(* IEC 61131-3 sources: programs/VI-54/VI-54_20171205/VI-54_20171205/Stations/PLC_VI54/VI-54_171014/Class/Camera_Master, 1 file *)

(* ---- Camera_Master.st ---- *)
(*!
<Class
	Name               = "Camera_Master"
	Revision           = "2.0"
	RealtimeTask       = "false"
	CyclicTask         = "false"
	BackgroundTask     = "false"
	Sigmatek           = "false"
	OSInterface        = "false"
	HighPriority       = "false"
	Automatic          = "false"
	UpdateMode         = "Prescan"
	SharedCommandTable = "true"
	Objectsize         = "(630,120)">
	<Channels>
		<Server Name="DataCompleted" Visualized="true" Initialize="false" WriteProtected="false" Retentive="false"/>
		<Server Name="IsOnline" Visualized="true" Initialize="false" WriteProtected="true" Retentive="false"/>
		<Server Name="NbrOfTriggers" Visualized="true" Initialize="false" WriteProtected="true" Retentive="false"/>
		<Server Name="SendCommand" Visualized="true" Initialize="false" WriteProtected="false" Retentive="false"/>
		<Server Name="TmrNewConnection" Visualized="true" Initialize="true" WriteProtected="false" Retentive="File"/>
		<Client Name="_TCPIP_CLIENT2" Required="true" Internal="true"/>
		<Client Name="cPort" Required="true" Internal="false" Comment="port number ... must be connected or initialized"/>
		<Client Name="iFc_Trigger" Required="true" Internal="false"/>
		<Client Name="IpAdres" Required="true" Internal="true"/>
	</Channels>
	<Separators>
		<Servers>
			<SepChn Position="3"/>
			<SepChn Position="5"/>
		</Servers>
	</Separators>
	<Network Name="Camera_Master">
		<!-- List of Components in this network -->
		<Components>
			<Object
				Name       = "_base"
				Class      = "MachineBase"
				Position   = "(218,120)"
				Visualized = "true">
				<Channels>
					<Server Name="ObjectServer"/>
					<Server Name="RunningMode"/>
					<Server Name="Stepper"/>
				</Channels>
			</Object>
			<Object
				Name           = "_TCPIP_CLIENT2"
				Class          = "_TCPIP_CLIENT"
				Position       = "(210,660)"
				Visualized     = "false"
				CyclicTime     = "10 ms"
				BackgroundTime = "always">
				<Channels>
					<Server Name="Control"/>
					<Server Name="SemaName01"/>
					<Server Name="SemaName02"/>
					<Server Name="TaskName"/>
					<Client Name="cConfig"/>
					<Client Name="cMaxConnections" Value="0"/>
					<Client Name="co_MultiTask"/>
					<Client Name="co_SigCLib"/>
					<Client Name="co_StdLib"/>
					<Client Name="co_Task"/>
					<Client Name="cPort" Value="500"/>
					<Client Name="cSizeOfTXBuffer"/>
				</Channels>
			</Object>
			<Object
				Name       = "IpAdres"
				Class      = "StringRAM"
				Position   = "(210,420)"
				Visualized = "true"
				Remotely   = "true">
				<Channels>
					<Server Name="Data" Value="&quot;10.10.150.26&quot;"/>
					<Client Name="SingleRealloc" Value="1"/>
					<Client Name="UseFile"/>
				</Channels>
			</Object>
		</Components>
		<Comments>
		</Comments>
		<!-- List of Connections in this network -->
		<Connections>
			<Connection Source="this.ObjectServer" Destination="_base.ObjectServer" Vertices="(1006,210),(834,210),"/>
			<Connection Source="this.Stepper" Destination="_base.Stepper" Vertices="(1006,270),(834,270),"/>
			<Connection Source="this.RunningMode" Destination="_base.RunningMode" Vertices="(1006,330),(834,330),"/>
			<Connection Source="this.IpAdres" Destination="IpAdres.Data"/>
			<Connection Source="this._TCPIP_CLIENT2" Destination="_TCPIP_CLIENT2.Control"/>
			<Connection Source="_TCPIP_CLIENT2.cPort" Destination="this.cPort" Vertices="(210,750),(38,390),"/>
		</Connections>
		<!-- Headerfiles -->
		<Options>
		</Options>
	</Network>
</Class>
*)
#pragma using MachineBase

Camera_Master : CLASS
: MachineBase
	TYPE
	  IpAdrStr : ARRAY [0..15] OF CHAR;
	  SendCommands :  //! <Type Public="true" Name="SendCommands"/>
	  (
	    eNoCommand,
	    eReboot,
	    eRestart,
	    eTrigger
	  )$UDINT;
#pragma pack(push, 1)
	  SendStr : STRUCT
	    HeartBeat : BOOL;
	    Command : SendCommands;
	  END_STRUCT;
#pragma pack(pop)
	END_TYPE
  //Servers:
	IsOnline 	: SvrCh_DINT;
	NbrOfTriggers 	: SvrCh_DINT;
	TmrNewConnection 	: SvrCh_UDINT;
	DataCompleted 	: SvrCh_DINT;
	SendCommand 	: SvrCh_SendCommands_PTofCls_Camera_Master;
  //Clients:
	IpAdres 	: CltChCmd_StringRAM;
	cPort 	: CltCh_DINT;
	_TCPIP_CLIENT2 	: CltChCmd__TCPIP_CLIENT;
	iFc_Trigger 	: CltChCmd_ProductTrigger;
  //Variables:
		Handle 	: DINT;
		Adress_TCP 	: IpAdrStr;
		CameraDataStr 	: CameraData;
		TmrDelay 	: UDINT;
		TmrHeartBeat 	: UDINT;
		CameraBits : BDINT
		[
		  1 SendStr,
		];

		SendData 	: SendStr;
  //Functions:

	FUNCTION VIRTUAL GLOBAL MyCyTask;

	FUNCTION GLOBAL MyCallBack
		VAR_INPUT
			pData 	: ^void;
			udSize 	: UDINT;
		END_VAR;

	FUNCTION GLOBAL GetData
		VAR_OUTPUT
			Ptr 	: CameraData;
		END_VAR;

	FUNCTION GLOBAL ResetData;

	FUNCTION GLOBAL gmSendData
		VAR_INPUT
			Data 	: ^void;
		END_VAR
		VAR_OUTPUT
			Retcode 	: BOOL;
		END_VAR;

	FUNCTION GLOBAL gmHeartBeat;

	FUNCTION GLOBAL gmTrigger;

	FUNCTION VIRTUAL GLOBAL SendCommand::Write
		VAR_INPUT
			input (EAX) 	: Camera_Master::SendCommands;
		END_VAR
		VAR_OUTPUT
			result (EAX) 	: Camera_Master::SendCommands;
		END_VAR;
  //Tables:
	FUNCTION @STD
		VAR_OUTPUT
			ret_code	: CONFSTATES;
		END_VAR;
	FUNCTION GLOBAL TAB @CT_;
END_CLASS;

#pragma using _TCPIP_CLIENT
#pragma using StringRAM
#pragma usingLtd ProductTrigger

FUNCTION VIRTUAL GLOBAL Camera_Master::MyCyTask

  _TCPIP_CLIENT2.CyWork(EAX:= 0);
  IsOnline := _TCPIP_CLIENT2.IsConnected(dHandle:= Handle);

  // Open methodes
  gmTrigger();
  gmHeartBeat();

  // Check for sending data
  if CameraBits.SendStr = true then
    if gmSendData(Data:= #SendData) = true then
      CameraBits.SendStr := False;
    end_if;
  end_if;

  case Stepper of
  00: // Check communication
    if IsOnline = false then
      Stepper += 1;
    end_if;

  01: // Make connection
    IpAdres.ReadDataOff(udOff:= 0, pData:= #Adress_TCP$Usint, udMax := sizeof(IpAdrStr));
    Adress_TCP[15] := cNul;
    Handle := _TCPIP_CLIENT2.AddConnection( pIPAddress    := "10.10.150.26",
                                            pCallbackThis := this,
                                            pCallbackMeth := #MyCallBack(),
                                            udTimeout     := 0);
    TmrDelay := ops.tAbsolute;
    Stepper += 1;

  02: // Check online state
    if IsOnline > 0 then
      TmrDelay := ops.tAbsolute;
    elsif (ops.tAbsolute - TmrDelay) >= TmrNewConnection then
      Stepper -= 1;
    end_if;
  end_case;

END_FUNCTION

FUNCTION GLOBAL Camera_Master::MyCallBack
	VAR_INPUT
		pData 	: ^void;
		udSize 	: UDINT;
	END_VAR

  // Set data into array
  _memset(dest:= #CameraDataStr, usByte:= 0, cntr:= sizeof(CameraData));
  _memcpy(ptr1:= #CameraDataStr, ptr2:= pData, cntr:= sizeof(CameraData));

  // Set bit that we receive new data
  DataCompleted := 1;

END_FUNCTION

FUNCTION GLOBAL Camera_Master::GetData
	VAR_OUTPUT
		Ptr 	: CameraData;
	END_VAR

  Ptr := CameraDataStr;

  // Reset data after reading
  ResetData();

END_FUNCTION

FUNCTION GLOBAL Camera_Master::ResetData

  // Reset all the data
  DataCompleted     := 0;

  // Reset pointer
  _memset(dest:= #CameraDataStr, usByte:= 0, cntr:= sizeof(CameraData));

END_FUNCTION

FUNCTION GLOBAL Camera_Master::gmHeartBeat

  // Every second a heartbeat
  if (ops.tAbsolute - TmrHeartBeat) >= 1000 then
    SendData.HeartBeat  := (SendData.HeartBeat XOR 1);
    CameraBits.SendStr  := true;
    TmrHeartBeat        := ops.tAbsolute;
  end_if;

END_FUNCTION

FUNCTION GLOBAL Camera_Master::gmTrigger

  // Set trigger offset
  iFc_Trigger.SetTriggerOffset(State:= (RecipePtr^.Camera.TriggerOffset * cIntUnitsTo_mm));

  // Check trigger
  if Standaard.R_TRIG(CLK:= iFc_Trigger.OffsetTrigger()) then
    SendData.Command   := SendCommands::eTrigger;
    CameraBits.SendStr := True;
  end_if;

END_FUNCTION

FUNCTION VIRTUAL GLOBAL Camera_Master::SendCommand::Write
	VAR_INPUT
		input (EAX) 	: Camera_Master::SendCommands;
	END_VAR
	VAR_OUTPUT
		result (EAX) 	: Camera_Master::SendCommands;
	END_VAR

	SendCommand := input;

  SendData.Command   := SendCommand;
  CameraBits.SendStr := True;
  SendCommand        := SendCommands::eNoCommand;

	result := SendCommand;

END_FUNCTION

FUNCTION GLOBAL Camera_Master::gmSendData
	VAR_INPUT
		Data 	: ^void;
	END_VAR
	VAR_OUTPUT
		Retcode 	: BOOL;
	END_VAR

  // Set ini
  Retcode := False;

  // Send data
  if _TCPIP_CLIENT2.SendData(pData:= Data, udSize:=sizeof(Data), dHandle:=Handle, bDirect:=true) = 0 then
    Retcode := True;
  end_if;

END_FUNCTION
